// TIA Portal V17 export
// export: Created 2024-08-20T11:47:33.1327124Z, ExportSetting WithDefaults, DisplayName Totally Integrated Automation Portal, DisplayVersion V17 Update 4, DisplayName TIA Portal Openness, DisplayVersion V17 Update 4, DisplayName TIA Portal Version Control Interface, DisplayVersion V17, DisplayName STEP 7 Professional, DisplayVersion V17 Update 4, DisplayName STEP 7 Safety, DisplayVersion V17, DisplayName WinCC Advanced, DisplayVersion V17 Update 4
DATA_BLOCK "ANALOGICOS_DB_1"   // DB5
VERSION : 0.1
// stored: AutoNumber true, DBAccessibleFromOPCUA true, InstanceOfName ANALOGICOS, InstanceOfType FB
"ANALOGICOS"
   // VAR
   //    LIT_001 { S7_SetPoint := 'True'} : "INSTRUMENTO";
   // END_VAR
BEGIN
END_DATA_BLOCK
